Omron CX-Programmer project NewProject (CX-Programmer 9.73)

# PLC NewPLC1: CP1E N30

## Global symbols (name address type ; comment)
0.03 BOOL  ; sensor produk
0.02 BOOL  ; sensor box
100.01 BOOL  ; conveyor produk
100.00 BOOL  ; conveyor box
0.00 BOOL  ; start
0.01 BOOL  ; stop

## Program NewProgram1 (cyclic task 0)

### Section Section1

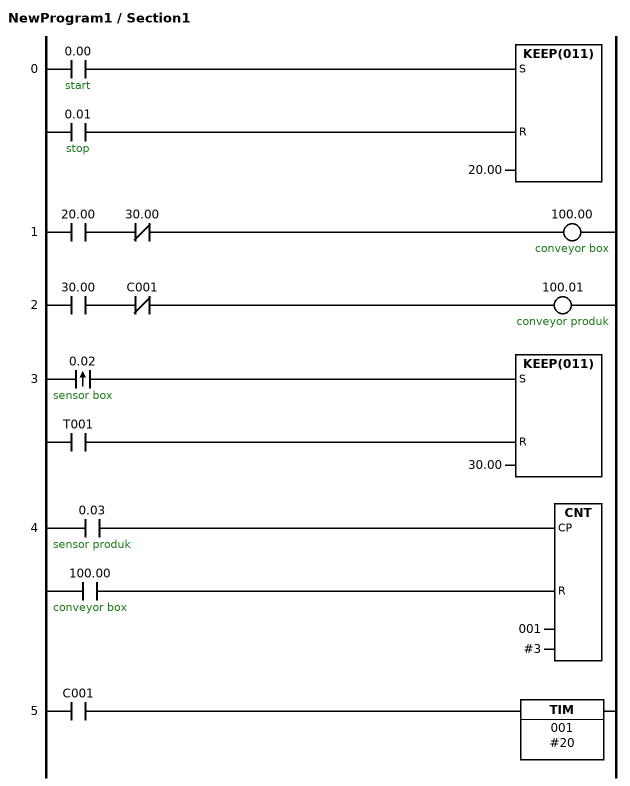
; rung 0
LD 0.00  ; start
LD 0.01  ; stop
KEEP(011) 20.00
; rung 1
LD 20.00
ANDNOT 30.00
OUT 100.00  ; conveyor box
; rung 2
LD 30.00
ANDNOT C001
OUT 100.01  ; conveyor produk
; rung 3
@LD 0.02  ; sensor box
LD T001
KEEP(011) 30.00
; rung 4
LD 0.03  ; sensor produk
LD 100.00  ; conveyor box
CNT 001 #3
; rung 5
LD C001
TIM 001 #20

### Section END
; rung 0
END(001)